Omron CX-Programmer project NewProject (CX-Programmer 9.61)

# PLC NewPLC1: CP1H X

## Global symbols (name address type ; comment)
10.01 BOOL  ; 2
0.00 BOOL  ; PB1
0.01 BOOL  ; PB2
0.02 BOOL  ; PB EMG
100.00 BOOL  ; SOL 1
100.01 BOOL  ; SOL 2
100.02 BOOL  ; SOL 1
100.03 BOOL  ; SOL 2
100.05 BOOL  ; pl1
101.00 BOOL  ; PL 2
101.01 BOOL  ; SOL 1-2
101.02 BOOL  ; SOL 1-1
101.03 BOOL  ; SOL 2-1
101.04 BOOL  ; SOL 2-2
10.00 BOOL  ; SOL 1
10.02 BOOL  ; SOL 3
10.03 BOOL  ; SOL 4
20.00 BOOL  ; PB 1
20.01 BOOL  ; PB 2
20.02 BOOL  ; PB EMG
30.00 BOOL  ; CR 1
30.01 BOOL  ; CR 2
5 CHANNEL  ; TIMER 1
T0001 BOOL  ; T1
T0002 BOOL  ; TIMER 2
T0003 BOOL  ; TIMER 3
T0004 BOOL  ; TIMER 4
T0005 BOOL  ; TIMER 5

## Program NewProgram1 (cyclic task 0)

### Section INPUT

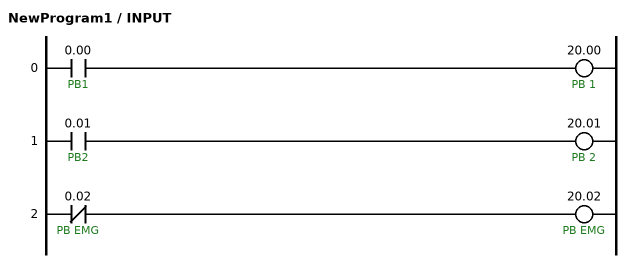
; rung 0
LD 0.00  ; PB1
OUT 20.00  ; PB 1
; rung 1
LD 0.01  ; PB2
OUT 20.01  ; PB 2
; rung 2
LDNOT 0.02  ; PB EMG
OUT 20.02  ; PB EMG

### Section OUTPUT

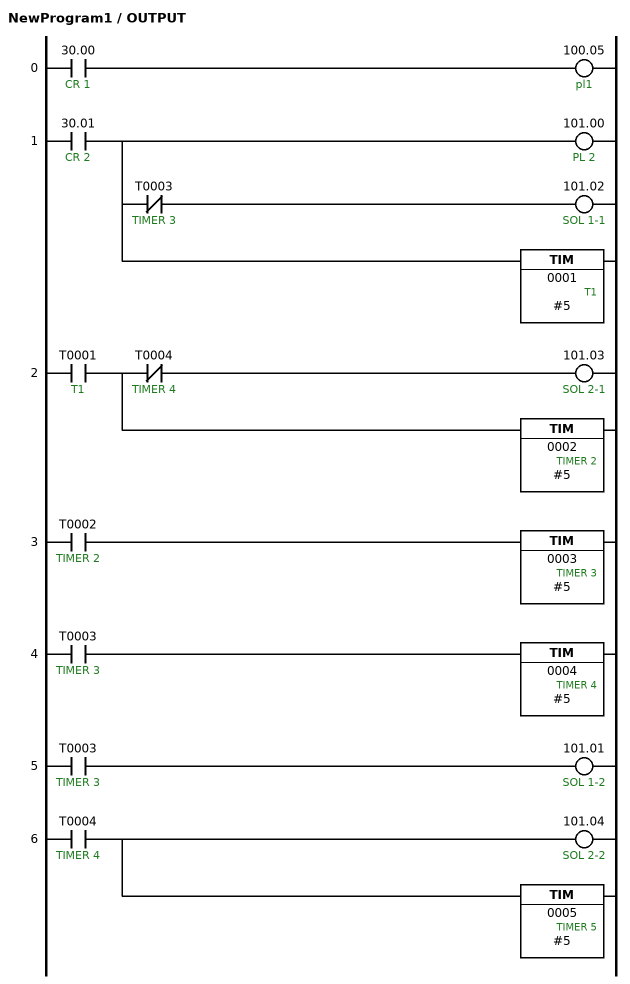
; rung 0
LD 30.00  ; CR 1
OUT 100.05  ; pl1
; rung 1
LD 30.01  ; CR 2
OUT TR0
OUT 101.00  ; PL 2
ANDNOT T0003  ; TIMER 3
OUT 101.02  ; SOL 1-1
LD TR0
TIM 0001 #5  ; T1
; rung 2
LD T0001  ; T1
OUT TR0
ANDNOT T0004  ; TIMER 4
OUT 101.03  ; SOL 2-1
LD TR0
TIM 0002 #5  ; TIMER 2
; rung 3
LD T0002  ; TIMER 2
TIM 0003 #5  ; TIMER 3
; rung 4
LD T0003  ; TIMER 3
TIM 0004 #5  ; TIMER 4
; rung 5
LD T0003  ; TIMER 3
OUT 101.01  ; SOL 1-2
; rung 6
LD T0004  ; TIMER 4
OUT 101.04  ; SOL 2-2
TIM 0005 #5  ; TIMER 5

### Section RANGKAIAN

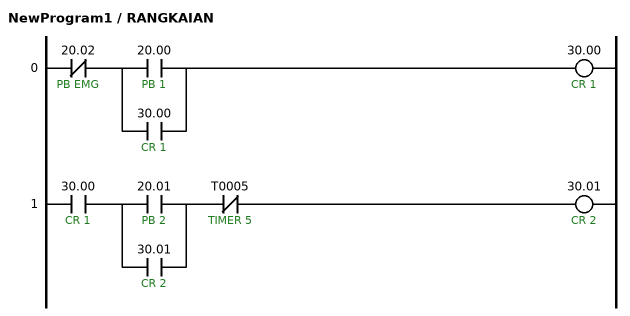
; rung 0
LDNOT 20.02  ; PB EMG
LD 20.00  ; PB 1
OR 30.00  ; CR 1
ANDLD
OUT 30.00  ; CR 1
; rung 1
LD 30.00  ; CR 1
LD 20.01  ; PB 2
OR 30.01  ; CR 2
ANDLD
ANDNOT T0005  ; TIMER 5
OUT 30.01  ; CR 2

### Section Section1

### Section END
; rung 0
END(001)